Staubli VAL3: IOInterface.pjx

--- IOInterface.pjx ---
Parameters version=s7.9.1 stackSize=5000 millimeterUnit=true
Program file=init.pgx
Program file=readAll.pgx
Program file=start.pgx
Program file=stop.pgx
Program file=writeSingle.pgx
Data file=IOInterface.dtx
Library alias=IOModule path=Disk://ros_libs/IOModule/IOModule.pjx autoload=true password=

--- IOInterface.dtx ---
public bool bBasicIO1
public bool bBasicIO2
dio diBasicIn[16]
  [0] = {link=BasicIO-1\%I0}
  [1] = {link=BasicIO-1\%I1}
  [2] = {link=BasicIO-1\%I2}
  [3] = {link=BasicIO-1\%I3}
  [4] = {link=BasicIO-1\%I4}
  [5] = {link=BasicIO-1\%I5}
  [6] = {link=BasicIO-1\%I6}
  [7] = {link=BasicIO-1\%I7}
  [8] = {link=BasicIO-1\%I8}
  [9] = {link=BasicIO-1\%I9}
  [10] = {link=BasicIO-1\%I10}
  [11] = {link=BasicIO-1\%I11}
  [12] = {link=BasicIO-1\%I12}
  [13] = {link=BasicIO-1\%I13}
  [14] = {link=BasicIO-1\%I14}
  [15] = {link=BasicIO-1\%I15}
dio diBasicIn2[16]
  [0] = {link=BasicIO-2\%I0}
  [1] = {link=BasicIO-2\%I1}
  [2] = {link=BasicIO-2\%I2}
  [3] = {link=BasicIO-2\%I3}
  [4] = {link=BasicIO-2\%I4}
  [5] = {link=BasicIO-2\%I5}
  [6] = {link=BasicIO-2\%I6}
  [7] = {link=BasicIO-2\%I7}
  [8] = {link=BasicIO-2\%I8}
  [9] = {link=BasicIO-2\%I9}
  [10] = {link=BasicIO-2\%I10}
  [11] = {link=BasicIO-2\%I11}
  [12] = {link=BasicIO-2\%I12}
  [13] = {link=BasicIO-2\%I13}
  [14] = {link=BasicIO-2\%I14}
  [15] = {link=BasicIO-2\%I15}
dio diBasicOut[16]
  [0] = {link=BasicIO-1\%Q0}
  [1] = {link=BasicIO-1\%Q1}
  [2] = {link=BasicIO-1\%Q2}
  [3] = {link=BasicIO-1\%Q3}
  [4] = {link=BasicIO-1\%Q4}
  [5] = {link=BasicIO-1\%Q5}
  [6] = {link=BasicIO-1\%Q6}
  [7] = {link=BasicIO-1\%Q7}
  [8] = {link=BasicIO-1\%Q8}
  [9] = {link=BasicIO-1\%Q9}
  [10] = {link=BasicIO-1\%Q10}
  [11] = {link=BasicIO-1\%Q11}
  [12] = {link=BasicIO-1\%Q12}
  [13] = {link=BasicIO-1\%Q13}
  [14] = {link=BasicIO-1\%Q14}
  [15] = {link=BasicIO-1\%Q15}
dio diBasicOut2[16]
  [0] = {link=BasicIO-2\%Q0}
  [1] = {link=BasicIO-2\%Q1}
  [2] = {link=BasicIO-2\%Q2}
  [3] = {link=BasicIO-2\%Q3}
  [4] = {link=BasicIO-2\%Q4}
  [5] = {link=BasicIO-2\%Q5}
  [6] = {link=BasicIO-2\%Q6}
  [7] = {link=BasicIO-2\%Q7}
  [8] = {link=BasicIO-2\%Q8}
  [9] = {link=BasicIO-2\%Q9}
  [10] = {link=BasicIO-2\%Q10}
  [11] = {link=BasicIO-2\%Q11}
  [12] = {link=BasicIO-2\%Q12}
  [13] = {link=BasicIO-2\%Q13}
  [14] = {link=BasicIO-2\%Q14}
  [15] = {link=BasicIO-2\%Q15}
dio diUserIn[2]
  [0] = {link=usrIn0}
  [1] = {link=usrIn1}
dio diValveOut[2]
  [0] = {link=valve1}
  [1] = {link=valve2}

--- init.pgx ---
public program init()
  local num l_nStatus
begin
  // Copyright (c) 2021, Institute for Factory Automation and Production Systems (FAPS)
  //
  // Licensed under the Apache License, Version 2.0 (the "License");
  // you may not use this file except in compliance with the License.
  // You may obtain a copy of the License at
  //
  //     http://www.apache.org/licenses/LICENSE-2.0
  //
  // Unless required by applicable law or agreed to in writing, software
  // distributed under the License is distributed on an "AS IS" BASIS,
  // WITHOUT WARRANTIES OR CONDITIONS OF ANY KIND, either express or implied.
  // See the License for the specific language governing permissions and
  // limitations under the License.


  logMsg("[INFO] Called IOInterface:init()")

  // init IOModule enum
  call IOModule:init()

  // check IO status of the BasicIO module
  l_nStatus = ioStatus(diBasicIn[0])
  if (l_nStatus >= 0)
    bBasicIO1=true
    logMsg("[INFO] BasicIO available (status: "+toString("", l_nStatus)+")")
  else
    bBasicIO1=false
    logMsg("[INFO] BasicIO not available (status: "+toString("", l_nStatus)+")")
  endIf

  // check IO status of the BasicIO-2 module
  l_nStatus = ioStatus(diBasicIn2[0])
  if (l_nStatus >= 0)
    bBasicIO2=true
    logMsg("[INFO] BasicIO-2 available (status: "+toString("", l_nStatus)+")")
  else
    bBasicIO2=false
    logMsg("[INFO] BasicIO-2 not available (status: "+toString("", l_nStatus)+")")
  endIf
end

--- readAll.pgx ---
public program readAll(num& x_nUserIn (dimensions=1), num& x_nValveOut (dimensions=1), num& x_nBasicIn (dimensions=1), num& x_nBasicOut (dimensions=1), num& x_nBasicIn2 (dimensions=1), num& x_nBasicOut2 (dimensions=1))
begin
  // Copyright (c) 2021, Institute for Factory Automation and Production Systems (FAPS)
  //
  // Licensed under the Apache License, Version 2.0 (the "License");
  // you may not use this file except in compliance with the License.
  // You may obtain a copy of the License at
  //
  //     http://www.apache.org/licenses/LICENSE-2.0
  //
  // Unless required by applicable law or agreed to in writing, software
  // distributed under the License is distributed on an "AS IS" BASIS,
  // WITHOUT WARRANTIES OR CONDITIONS OF ANY KIND, either express or implied.
  // See the License for the specific language governing permissions and
  // limitations under the License.


  x_nUserIn=dioGet(diUserIn)
  x_nValveOut=dioGet(diValveOut)

  if (bBasicIO1)
    x_nBasicIn=dioGet(diBasicIn)
    x_nBasicOut=dioGet(diBasicOut)
  else
    x_nBasicIn=0
    x_nBasicOut=0
  endIf

  if (bBasicIO2)
    x_nBasicIn2=dioGet(diBasicIn)
    x_nBasicOut2=dioGet(diBasicOut)
  else
    x_nBasicIn2=0
    x_nBasicOut2=0
  endIf

end

--- stop.pgx ---
program stop()
begin
  // Copyright (c) 2021, Institute for Factory Automation and Production Systems (FAPS)
  //
  // Licensed under the Apache License, Version 2.0 (the "License");
  // you may not use this file except in compliance with the License.
  // You may obtain a copy of the License at
  //
  //     http://www.apache.org/licenses/LICENSE-2.0
  //
  // Unless required by applicable law or agreed to in writing, software
  // distributed under the License is distributed on an "AS IS" BASIS,
  // WITHOUT WARRANTIES OR CONDITIONS OF ANY KIND, either express or implied.
  // See the License for the specific language governing permissions and
  // limitations under the License.


end

--- writeSingle.pgx ---
public program writeSingle(num x_nModuleId (dimensions=1), num x_nPin (dimensions=1), bool x_bState (dimensions=1), bool& x_bSuccess (dimensions=1))
  local dio l_diSignal
  local num l_nPins
begin
  // Copyright (c) 2021, Institute for Factory Automation and Production Systems (FAPS)
  //
  // Licensed under the Apache License, Version 2.0 (the "License");
  // you may not use this file except in compliance with the License.
  // You may obtain a copy of the License at
  //
  //     http://www.apache.org/licenses/LICENSE-2.0
  //
  // Unless required by applicable law or agreed to in writing, software
  // distributed under the License is distributed on an "AS IS" BASIS,
  // WITHOUT WARRANTIES OR CONDITIONS OF ANY KIND, either express or implied.
  // See the License for the specific language governing permissions and
  // limitations under the License.


  x_bSuccess=true

  // get max pin count for given module
  switch x_nModuleId
    case IOModule:USER_IN,IOModule:VALVE_OUT
      l_nPins=2
    break
    case IOModule:BASIC_IN,IOModule:BASIC_OUT,IOModule:BASIC_IN_2,IOModule:BASIC_OUT_2
      l_nPins=16
    break
    default
      x_bSuccess=false
    break
  endSwitch

  // return if unknown module id was given
  if (x_bSuccess==false)
    popUpMsg("Error! Unknown module id: "+toString("",x_nModuleId))
    return
  endIf

  // check if pin index is out of range
  if (x_nPin>=l_nPins)
    popUpMsg("Error! Trying to set pin "+toString("",x_nPin)+" of module "+toString("",x_nModuleId))
    x_bSuccess=false
    return
  endIf

  // link signal source to local variable if possible
  switch x_nModuleId
    case IOModule:USER_IN
      dioLink(l_diSignal,diUserIn[x_nPin])
    break
    case IOModule:VALVE_OUT
      dioLink(l_diSignal,diValveOut[x_nPin])
    break
    case IOModule:BASIC_IN
      if (bBasicIO1)
        dioLink(l_diSignal,diBasicIn[x_nPin])
      else
        x_bSuccess=false
      endIf
    break
    case IOModule:BASIC_OUT
      if (bBasicIO1)
        dioLink(l_diSignal,diBasicOut[x_nPin])
      else
        x_bSuccess=false
      endIf
    break
    case IOModule:BASIC_IN_2
      if (bBasicIO2)
        dioLink(l_diSignal,diBasicIn2[x_nPin])
      else
        x_bSuccess=false
      endIf
    break
    case IOModule:BASIC_OUT_2
      if (bBasicIO2)
        dioLink(l_diSignal,diBasicOut2[x_nPin])
      else
        x_bSuccess=false
      endIf
    break
  endSwitch

  // set dio if linked successfully
  if (x_bSuccess)
    l_diSignal=x_bState
  endIf

end
